// TIA Portal V17 export
// export: Created 2024-08-29T18:23:46.9031876Z, ExportSetting WithDefaults, DisplayName Totally Integrated Automation Portal, DisplayVersion V17 Update 7, DisplayName TIA Portal Openness, DisplayVersion V17 Update 7, DisplayName TIA Portal Version Control Interface, DisplayVersion V17, DisplayName SINAMICS Startdrive Advanced, DisplayVersion V17 SP2, DisplayName SINAMICS Startdrive G110M, G120, G120C, G120D, G120P, G115D, DisplayVersion V17 SP2, DisplayName SINAMICS Startdrive G130, G150, S120, S150, SINAMICS MV, S210, DisplayVersion V17 SP2, DisplayName STEP 7 Professional, DisplayVersion V17 Update 7, DisplayName STEP 7 Safety, DisplayVersion V17 Update 6, DisplayName WinCC Advanced / Unified PC, DisplayVersion V17 Update 7
FUNCTION "miscelaneous" : Void   // FC5, LAD
{ S7_Optimized_Access := 'TRUE' }
VERSION : 0.1
// stored: AutoNumber true, IsIECCheckEnabled false, SetENOAutomatically false, UDAEnableTagReadback false
   VAR_TEMP
      INTERMITENTE : Bool;
      RESETEADO : Bool;
      RESULT_2 : UInt;
      Result_3 : Int;
   END_VAR
   VAR_TEMP   // added for the SCL form of the ladder/FBD networks
      _w1 : Bool;
      _w2 : Bool;
      _w3 : Bool;
      _w4 : Bool;
   END_VAR
BEGIN

REGION Network 1: HMI OPTIONS BUTTON SHUTOFF
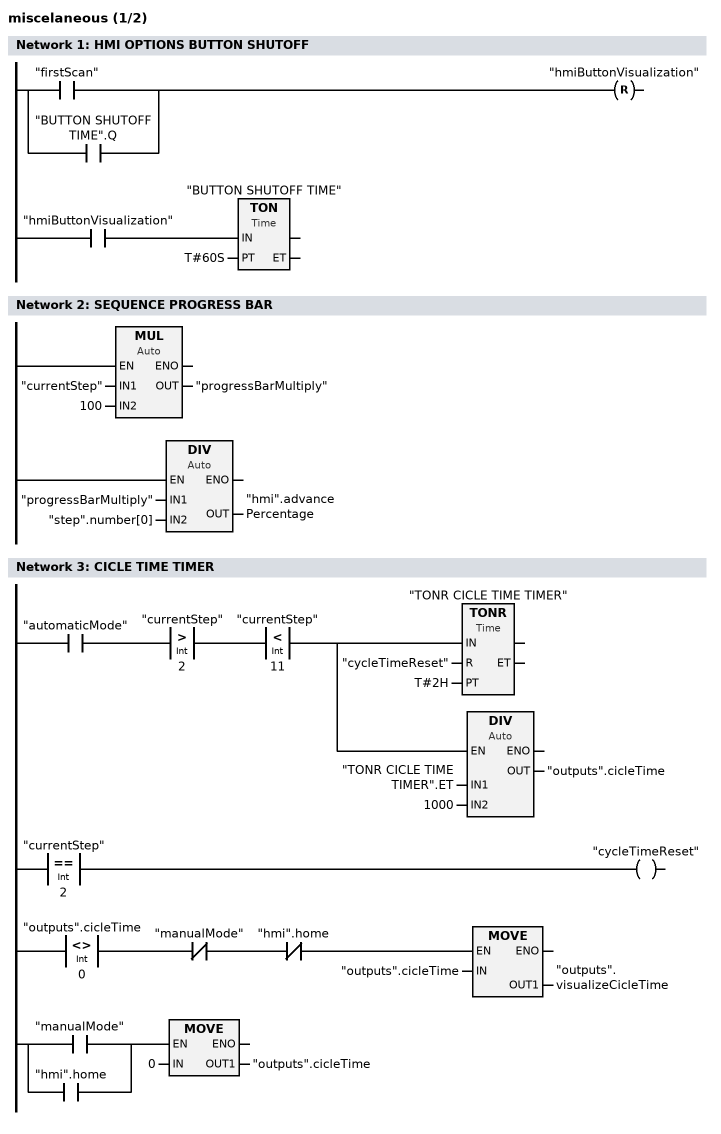
   RUNG wire#powerrail
      Contact( "firstScan" )
      wire#w1
      R_Coil( "hmiButtonVisualization" )
   END_RUNG
   RUNG wire#powerrail
      Contact( "BUTTON SHUTOFF TIME".Q )
   END_RUNG wire#w1
   RUNG wire#powerrail
      Contact( "hmiButtonVisualization" )
      { S7_Templates := "time_type := Time" } "BUTTON SHUTOFF TIME".TON(pt := T#60S, et =>)
   END_RUNG
   // the same network as SCL:
   IF "firstScan" OR "BUTTON SHUTOFF TIME".Q THEN "hmiButtonVisualization" := FALSE; END_IF;
   "BUTTON SHUTOFF TIME".TON(IN := "hmiButtonVisualization", PT := T#60S);
END_REGION

REGION Network 2: SEQUENCE PROGRESS BAR
   RUNG wire#powerrail
      Mul(in1 := "currentStep", in2 := 100, out => "progressBarMultiply")
   END_RUNG
   RUNG wire#powerrail
      Div(in1 := "progressBarMultiply", in2 := "step".number[0], out => "hmi".advancePercentage)
   END_RUNG
   // the same network as SCL:
   "progressBarMultiply" := "currentStep" * 100;
   "hmi".advancePercentage := "progressBarMultiply" / "step".number[0];
END_REGION

REGION Network 3: CICLE TIME TIMER
   RUNG wire#powerrail
      Contact( "automaticMode" )
      { S7_Templates := "SrcType := Int" } GT_Contact(in1 := "currentStep", in2 := 2)
      { S7_Templates := "SrcType := Int" } LT_Contact(in1 := "currentStep", in2 := 11)
      wire#w1
      { S7_Templates := "time_type := Time" } "TONR CICLE TIME TIMER".TONR(r := "cycleTimeReset", pt := T#2H, et =>)
   END_RUNG
   RUNG wire#w1
      Div(in1 := "TONR CICLE TIME TIMER".ET, in2 := 1000, out => "outputs".cicleTime)
   END_RUNG
   RUNG wire#powerrail
      { S7_Templates := "SrcType := Int" } EQ_Contact(in1 := "currentStep", in2 := 2)
      Coil( "cycleTimeReset" )
   END_RUNG
   RUNG wire#powerrail
      { S7_Templates := "SrcType := Int" } NE_Contact(in1 := "outputs".cicleTime, in2 := 0)
      I_Contact( "manualMode" )
      I_Contact( "hmi".home )
      Move(in := "outputs".cicleTime, out1 => "outputs".visualizeCicleTime)
   END_RUNG
   RUNG wire#powerrail
      Contact( "manualMode" )
      wire#w2
      Move(in := 0, out1 => "outputs".cicleTime)
   END_RUNG
   RUNG wire#powerrail
      Contact( "hmi".home )
   END_RUNG wire#w2
   // the same network as SCL:
   #_w1 := "automaticMode" AND ("currentStep" > 2) AND ("currentStep" < 11);
   "TONR CICLE TIME TIMER".TONR(IN := #_w1, R := "cycleTimeReset", PT := T#2H);
   IF #_w1 THEN "outputs".cicleTime := "TONR CICLE TIME TIMER".ET / 1000; END_IF;
   "cycleTimeReset" := "currentStep" = 2;
   IF ("outputs".cicleTime <> 0) AND NOT "manualMode" AND NOT "hmi".home THEN
       "outputs".visualizeCicleTime := "outputs".cicleTime;
   END_IF;
   IF "manualMode" OR "hmi".home THEN "outputs".cicleTime := 0; END_IF;
END_REGION

REGION Network 4: STEP CHANGE TIMER
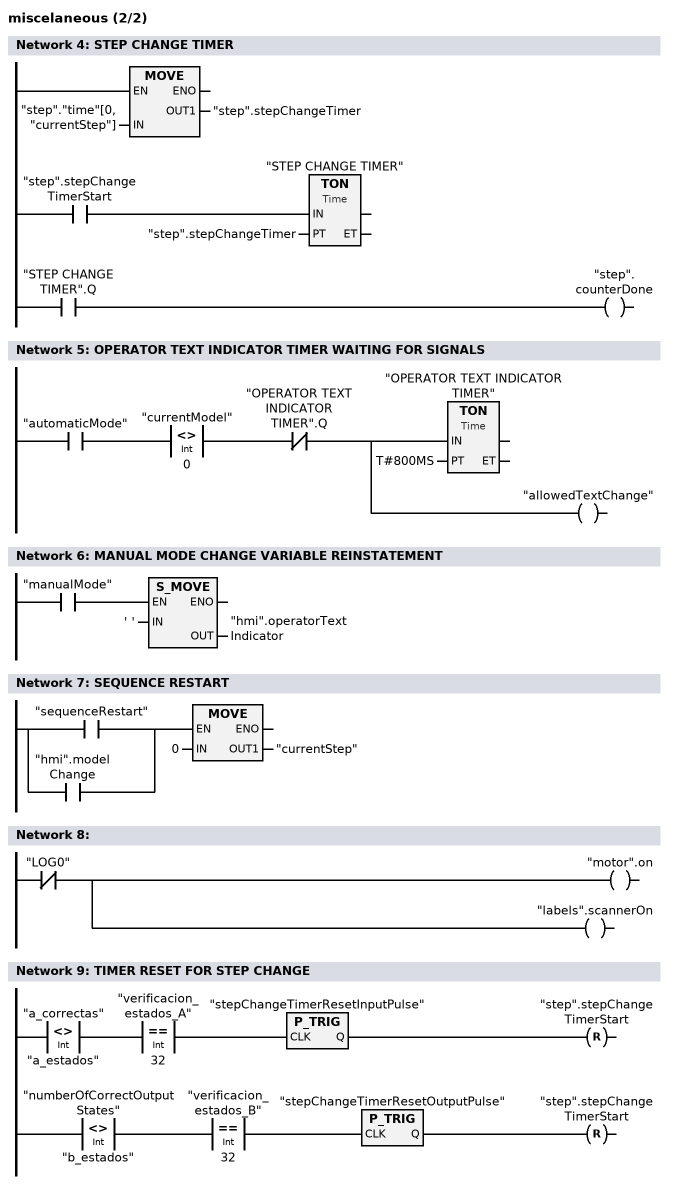
   RUNG wire#powerrail
      Move(in := "step"."time"[0, "currentStep"], out1 => "step".stepChangeTimer)
   END_RUNG
   RUNG wire#powerrail
      Contact( "step".stepChangeTimerStart )
      { S7_Templates := "time_type := Time" } "STEP CHANGE TIMER".TON(pt := "step".stepChangeTimer, et =>)
   END_RUNG
   RUNG wire#powerrail
      Contact( "STEP CHANGE TIMER".Q )
      Coil( "step".counterDone )
   END_RUNG
   // the same network as SCL:
   "step".stepChangeTimer := "step"."time"[0, "currentStep"];
   "STEP CHANGE TIMER".TON(IN := "step".stepChangeTimerStart, PT := "step".stepChangeTimer);
   "step".counterDone := "STEP CHANGE TIMER".Q;
END_REGION

REGION Network 5: OPERATOR TEXT INDICATOR TIMER WAITING FOR SIGNALS
   RUNG wire#powerrail
      Contact( "automaticMode" )
      { S7_Templates := "SrcType := Int" } NE_Contact(in1 := "currentModel", in2 := 0)
      I_Contact( "OPERATOR TEXT INDICATOR TIMER".Q )
      wire#w1
      { S7_Templates := "time_type := Time" } "OPERATOR TEXT INDICATOR TIMER".TON(pt := T#800MS, et =>)
   END_RUNG
   RUNG wire#w1
      Coil( "allowedTextChange" )
   END_RUNG
   // the same network as SCL:
   #_w1 := "automaticMode" AND ("currentModel" <> 0) AND NOT "OPERATOR TEXT INDICATOR TIMER".Q;
   "OPERATOR TEXT INDICATOR TIMER".TON(IN := #_w1, PT := T#800MS);
   "allowedTextChange" := #_w1;
END_REGION

REGION Network 6: MANUAL MODE CHANGE VARIABLE REINSTATEMENT
   RUNG wire#powerrail
      Contact( "manualMode" )
      S_Move(in := ' ', out => "hmi".operatorTextIndicator)
   END_RUNG
   // the same network as SCL:
   IF "manualMode" THEN "hmi".operatorTextIndicator := ' '; END_IF;
END_REGION

REGION Network 7: SEQUENCE RESTART
   RUNG wire#powerrail
      Contact( "sequenceRestart" )
      wire#w1
      Move(in := 0, out1 => "currentStep")
   END_RUNG
   RUNG wire#powerrail
      Contact( "hmi".modelChange )
   END_RUNG wire#w1
   // the same network as SCL:
   IF "sequenceRestart" OR "hmi".modelChange THEN "currentStep" := 0; END_IF;
END_REGION

REGION Network 8
   RUNG wire#powerrail
      I_Contact( "LOG0" )
      wire#w1
      Coil( "motor".on )
   END_RUNG
   RUNG wire#w1
      Coil( "labels".scannerOn )
   END_RUNG
   // the same network as SCL:
   "motor".on := NOT "LOG0";
   "labels".scannerOn := NOT "LOG0";
END_REGION

REGION Network 9: TIMER RESET FOR STEP CHANGE
   RUNG wire#powerrail
      { S7_Templates := "SrcType := Int" } NE_Contact(in1 := "a_correctas", in2 := "a_estados")
      { S7_Templates := "SrcType := Int" } EQ_Contact(in1 := "verificacion_estados_A", in2 := 32)
      P_Trig( "stepChangeTimerResetInputPulse" )
      R_Coil( "step".stepChangeTimerStart )
   END_RUNG
   RUNG wire#powerrail
      { S7_Templates := "SrcType := Int" } NE_Contact(in1 := "numberOfCorrectOutputStates", in2 := "b_estados")
      { S7_Templates := "SrcType := Int" } EQ_Contact(in1 := "verificacion_estados_B", in2 := 32)
      P_Trig( "stepChangeTimerResetOutputPulse" )
      R_Coil( "step".stepChangeTimerStart )
   END_RUNG
   // the same network as SCL:
   #_w1 := ("a_correctas" <> "a_estados") AND ("verificacion_estados_A" = 32);
   #_w2 := #_w1 AND NOT "stepChangeTimerResetInputPulse";   // rising edge
   "stepChangeTimerResetInputPulse" := #_w1;
   IF #_w2 THEN "step".stepChangeTimerStart := FALSE; END_IF;
   #_w3 := ("numberOfCorrectOutputStates" <> "b_estados") AND ("verificacion_estados_B" = 32);
   #_w4 := #_w3 AND NOT "stepChangeTimerResetOutputPulse";   // rising edge
   "stepChangeTimerResetOutputPulse" := #_w3;
   IF #_w4 THEN "step".stepChangeTimerStart := FALSE; END_IF;
END_REGION
END_FUNCTION
